									[9].arrDataOut[60]	:=	<0, 8, 0>TIIB(104)^API^Data^io^Outputs^Request Data[30];
									[9].arrDataOut[61]	:=	<0, 8, 8>TIIB(104)^API^Data^io^Outputs^Request Data[30];
									[9].arrDataOut[62]	:=	<0, 8, 0>TIIB(104)^API^Data^io^Outputs^Request Data[31];
									[9].arrDataOut[63]	:=	<0, 8, 8>TIIB(104)^API^Data^io^Outputs^Request Data[31];
									[9].PnIoBoxState 	:=	<0, 16, 0>TIIB(104)^Inputs^PnIoBoxState;
									[10].arrDataIn[0]	:=	<0, 8, 0>TIIB(105)^API^Data^io^Inputs^Response Data[0];
									[10].arrDataIn[1]	:=	<0, 8, 8>TIIB(105)^API^Data^io^Inputs^Response Data[0];
									[10].arrDataIn[2]	:=	<0, 8, 0>TIIB(105)^API^Data^io^Inputs^Response Data[1];
									[10].arrDataIn[3]	:=	<0, 8, 8>TIIB(105)^API^Data^io^Inputs^Response Data[1];
									[10].arrDataIn[4]	:=	<0, 8, 0>TIIB(105)^API^Data^io^Inputs^Response Data[2];
									[10].arrDataIn[5]	:=	<0, 8, 8>TIIB(105)^API^Data^io^Inputs^Response Data[2];
									[10].arrDataIn[6]	:=	<0, 8, 0>TIIB(105)^API^Data^io^Inputs^Response Data[3];
									[10].arrDataIn[7]	:=	<0, 8, 8>TIIB(105)^API^Data^io^Inputs^Response Data[3];
									[10].arrDataIn[8]	:=	<0, 8, 0>TIIB(105)^API^Data^io^Inputs^Response Data[4];
									[10].arrDataIn[9]	:=	<0, 8, 8>TIIB(105)^API^Data^io^Inputs^Response Data[4];
									[10].arrDataIn[10]	:=	<0, 8, 0>TIIB(105)^API^Data^io^Inputs^Response Data[5];
									[10].arrDataIn[11]	:=	<0, 8, 8>TIIB(105)^API^Data^io^Inputs^Response Data[5];
									[10].arrDataIn[12]	:=	<0, 8, 0>TIIB(105)^API^Data^io^Inputs^Response Data[6];
									[10].arrDataIn[13]	:=	<0, 8, 8>TIIB(105)^API^Data^io^Inputs^Response Data[6];
									[10].arrDataIn[14]	:=	<0, 8, 0>TIIB(105)^API^Data^io^Inputs^Response Data[7];
									[10].arrDataIn[15]	:=	<0, 8, 8>TIIB(105)^API^Data^io^Inputs^Response Data[7];
									[10].arrDataIn[16]	:=	<0, 8, 0>TIIB(105)^API^Data^io^Inputs^Response Data[8];
									[10].arrDataIn[17]	:=	<0, 8, 8>TIIB(105)^API^Data^io^Inputs^Response Data[8];
									[10].arrDataIn[18]	:=	<0, 8, 0>TIIB(105)^API^Data^io^Inputs^Response Data[9];
									[10].arrDataIn[19]	:=	<0, 8, 8>TIIB(105)^API^Data^io^Inputs^Response Data[9];
									[10].arrDataIn[20]	:=	<0, 8, 0>TIIB(105)^API^Data^io^Inputs^Response Data[10];
									[10].arrDataIn[21]	:=	<0, 8, 8>TIIB(105)^API^Data^io^Inputs^Response Data[10];
									[10].arrDataIn[22]	:=	<0, 8, 0>TIIB(105)^API^Data^io^Inputs^Response Data[11];
									[10].arrDataIn[23]	:=	<0, 8, 8>TIIB(105)^API^Data^io^Inputs^Response Data[11];
									[10].arrDataIn[24]	:=	<0, 8, 0>TIIB(105)^API^Data^io^Inputs^Response Data[12];
									[10].arrDataIn[25]	:=	<0, 8, 8>TIIB(105)^API^Data^io^Inputs^Response Data[12];
									[10].arrDataIn[26]	:=	<0, 8, 0>TIIB(105)^API^Data^io^Inputs^Response Data[13];
									[10].arrDataIn[27]	:=	<0, 8, 8>TIIB(105)^API^Data^io^Inputs^Response Data[13];
									[10].arrDataIn[28]	:=	<0, 8, 0>TIIB(105)^API^Data^io^Inputs^Response Data[14];
									[10].arrDataIn[29]	:=	<0, 8, 8>TIIB(105)^API^Data^io^Inputs^Response Data[14];
									[10].arrDataIn[30]	:=	<0, 8, 0>TIIB(105)^API^Data^io^Inputs^Response Data[15];
									[10].arrDataIn[31]	:=	<0, 8, 8>TIIB(105)^API^Data^io^Inputs^Response Data[15];
									[10].arrDataIn[32]	:=	<0, 8, 0>TIIB(105)^API^Data^io^Inputs^Response Data[16];
									[10].arrDataIn[33]	:=	<0, 8, 8>TIIB(105)^API^Data^io^Inputs^Response Data[16];
									[10].arrDataIn[34]	:=	<0, 8, 0>TIIB(105)^API^Data^io^Inputs^Response Data[17];
									[10].arrDataIn[35]	:=	<0, 8, 8>TIIB(105)^API^Data^io^Inputs^Response Data[17];
									[10].arrDataIn[36]	:=	<0, 8, 0>TIIB(105)^API^Data^io^Inputs^Response Data[18];
									[10].arrDataIn[37]	:=	<0, 8, 8>TIIB(105)^API^Data^io^Inputs^Response Data[18];
									[10].arrDataIn[38]	:=	<0, 8, 0>TIIB(105)^API^Data^io^Inputs^Response Data[19];
									[10].arrDataIn[39]	:=	<0, 8, 8>TIIB(105)^API^Data^io^Inputs^Response Data[19];
									[10].arrDataIn[40]	:=	<0, 8, 0>TIIB(105)^API^Data^io^Inputs^Response Data[20];
									[10].arrDataIn[41]	:=	<0, 8, 8>TIIB(105)^API^Data^io^Inputs^Response Data[20];
									[10].arrDataIn[42]	:=	<0, 8, 0>TIIB(105)^API^Data^io^Inputs^Response Data[21];
									[10].arrDataIn[43]	:=	<0, 8, 8>TIIB(105)^API^Data^io^Inputs^Response Data[21];
									[10].arrDataIn[44]	:=	<0, 8, 0>TIIB(105)^API^Data^io^Inputs^Response Data[22];
									[10].arrDataIn[45]	:=	<0, 8, 8>TIIB(105)^API^Data^io^Inputs^Response Data[22];
									[10].arrDataIn[46]	:=	<0, 8, 0>TIIB(105)^API^Data^io^Inputs^Response Data[23];
									[10].arrDataIn[47]	:=	<0, 8, 8>TIIB(105)^API^Data^io^Inputs^Response Data[23];
									[10].arrDataIn[48]	:=	<0, 8, 0>TIIB(105)^API^Data^io^Inputs^Response Data[24];
									[10].arrDataIn[49]	:=	<0, 8, 8>TIIB(105)^API^Data^io^Inputs^Response Data[24];
									[10].arrDataIn[50]	:=	<0, 8, 0>TIIB(105)^API^Data^io^Inputs^Response Data[25];
									[10].arrDataIn[51]	:=	<0, 8, 8>TIIB(105)^API^Data^io^Inputs^Response Data[25];
									[10].arrDataIn[52]	:=	<0, 8, 0>TIIB(105)^API^Data^io^Inputs^Response Data[26];
									[10].arrDataIn[53]	:=	<0, 8, 8>TIIB(105)^API^Data^io^Inputs^Response Data[26];
									[10].arrDataIn[54]	:=	<0, 8, 0>TIIB(105)^API^Data^io^Inputs^Response Data[27];
									[10].arrDataIn[55]	:=	<0, 8, 8>TIIB(105)^API^Data^io^Inputs^Response Data[27];
									[10].arrDataIn[56]	:=	<0, 8, 0>TIIB(105)^API^Data^io^Inputs^Response Data[28];
									[10].arrDataIn[57]	:=	<0, 8, 8>TIIB(105)^API^Data^io^Inputs^Response Data[28];
									[10].arrDataIn[58]	:=	<0, 8, 0>TIIB(105)^API^Data^io^Inputs^Response Data[29];
									[10].arrDataIn[59]	:=	<0, 8, 8>TIIB(105)^API^Data^io^Inputs^Response Data[29];
									[10].arrDataIn[60]	:=	<0, 8, 0>TIIB(105)^API^Data^io^Inputs^Response Data[30];
									[10].arrDataIn[61]	:=	<0, 8, 8>TIIB(105)^API^Data^io^Inputs^Response Data[30];
									[10].arrDataIn[62]	:=	<0, 8, 0>TIIB(105)^API^Data^io^Inputs^Response Data[31];
									[10].arrDataIn[63]	:=	<0, 8, 8>TIIB(105)^API^Data^io^Inputs^Response Data[31];
									[10].arrDataOut[0]	:=	<0, 8, 0>TIIB(105)^API^Data^io^Outputs^Request Data[0];
									[10].arrDataOut[1]	:=	<0, 8, 8>TIIB(105)^API^Data^io^Outputs^Request Data[0];
									[10].arrDataOut[2]	:=	<0, 8, 0>TIIB(105)^API^Data^io^Outputs^Request Data[1];
									[10].arrDataOut[3]	:=	<0, 8, 8>TIIB(105)^API^Data^io^Outputs^Request Data[1];
									[10].arrDataOut[4]	:=	<0, 8, 0>TIIB(105)^API^Data^io^Outputs^Request Data[2];
									[10].arrDataOut[5]	:=	<0, 8, 8>TIIB(105)^API^Data^io^Outputs^Request Data[2];
									[10].arrDataOut[6]	:=	<0, 8, 0>TIIB(105)^API^Data^io^Outputs^Request Data[3];
									[10].arrDataOut[7]	:=	<0, 8, 8>TIIB(105)^API^Data^io^Outputs^Request Data[3];
									[10].arrDataOut[8]	:=	<0, 8, 0>TIIB(105)^API^Data^io^Outputs^Request Data[4];
									[10].arrDataOut[9]	:=	<0, 8, 8>TIIB(105)^API^Data^io^Outputs^Request Data[4];
									[10].arrDataOut[10]	:=	<0, 8, 0>TIIB(105)^API^Data^io^Outputs^Request Data[5];
									[10].arrDataOut[11]	:=	<0, 8, 8>TIIB(105)^API^Data^io^Outputs^Request Data[5];
									[10].arrDataOut[12]	:=	<0, 8, 0>TIIB(105)^API^Data^io^Outputs^Request Data[6];
									[10].arrDataOut[13]	:=	<0, 8, 8>TIIB(105)^API^Data^io^Outputs^Request Data[6];
									[10].arrDataOut[14]	:=	<0, 8, 0>TIIB(105)^API^Data^io^Outputs^Request Data[7];
									[10].arrDataOut[15]	:=	<0, 8, 8>TIIB(105)^API^Data^io^Outputs^Request Data[7];
									[10].arrDataOut[16]	:=	<0, 8, 0>TIIB(105)^API^Data^io^Outputs^Request Data[8];
									[10].arrDataOut[17]	:=	<0, 8, 8>TIIB(105)^API^Data^io^Outputs^Request Data[8];
									[10].arrDataOut[18]	:=	<0, 8, 0>TIIB(105)^API^Data^io^Outputs^Request Data[9];
									[10].arrDataOut[19]	:=	<0, 8, 8>TIIB(105)^API^Data^io^Outputs^Request Data[9];
									[10].arrDataOut[20]	:=	<0, 8, 0>TIIB(105)^API^Data^io^Outputs^Request Data[10];
									[10].arrDataOut[21]	:=	<0, 8, 8>TIIB(105)^API^Data^io^Outputs^Request Data[10];
									[10].arrDataOut[22]	:=	<0, 8, 0>TIIB(105)^API^Data^io^Outputs^Request Data[11];
									[10].arrDataOut[23]	:=	<0, 8, 8>TIIB(105)^API^Data^io^Outputs^Request Data[11];
									[10].arrDataOut[24]	:=	<0, 8, 0>TIIB(105)^API^Data^io^Outputs^Request Data[12];
									[10].arrDataOut[25]	:=	<0, 8, 8>TIIB(105)^API^Data^io^Outputs^Request Data[12];
									[10].arrDataOut[26]	:=	<0, 8, 0>TIIB(105)^API^Data^io^Outputs^Request Data[13];
									[10].arrDataOut[27]	:=	<0, 8, 8>TIIB(105)^API^Data^io^Outputs^Request Data[13];
									[10].arrDataOut[28]	:=	<0, 8, 0>TIIB(105)^API^Data^io^Outputs^Request Data[14];
									[10].arrDataOut[29]	:=	<0, 8, 8>TIIB(105)^API^Data^io^Outputs^Request Data[14];
									[10].arrDataOut[30]	:=	<0, 8, 0>TIIB(105)^API^Data^io^Outputs^Request Data[15];
									[10].arrDataOut[31]	:=	<0, 8, 8>TIIB(105)^API^Data^io^Outputs^Request Data[15];
									[10].arrDataOut[32]	:=	<0, 8, 0>TIIB(105)^API^Data^io^Outputs^Request Data[16];
									[10].arrDataOut[33]	:=	<0, 8, 8>TIIB(105)^API^Data^io^Outputs^Request Data[16];
									[10].arrDataOut[34]	:=	<0, 8, 0>TIIB(105)^API^Data^io^Outputs^Request Data[17];
									[10].arrDataOut[35]	:=	<0, 8, 8>TIIB(105)^API^Data^io^Outputs^Request Data[17];
									[10].arrDataOut[36]	:=	<0, 8, 0>TIIB(105)^API^Data^io^Outputs^Request Data[18];
									[10].arrDataOut[37]	:=	<0, 8, 8>TIIB(105)^API^Data^io^Outputs^Request Data[18];
									[10].arrDataOut[38]	:=	<0, 8, 0>TIIB(105)^API^Data^io^Outputs^Request Data[19];
									[10].arrDataOut[39]	:=	<0, 8, 8>TIIB(105)^API^Data^io^Outputs^Request Data[19];
									[10].arrDataOut[40]	:=	<0, 8, 0>TIIB(105)^API^Data^io^Outputs^Request Data[20];
									[10].arrDataOut[41]	:=	<0, 8, 8>TIIB(105)^API^Data^io^Outputs^Request Data[20];
									[10].arrDataOut[42]	:=	<0, 8, 0>TIIB(105)^API^Data^io^Outputs^Request Data[21];
									[10].arrDataOut[43]	:=	<0, 8, 8>TIIB(105)^API^Data^io^Outputs^Request Data[21];
									[10].arrDataOut[44]	:=	<0, 8, 0>TIIB(105)^API^Data^io^Outputs^Request Data[22];
									[10].arrDataOut[45]	:=	<0, 8, 8>TIIB(105)^API^Data^io^Outputs^Request Data[22];
									[10].arrDataOut[46]	:=	<0, 8, 0>TIIB(105)^API^Data^io^Outputs^Request Data[23];
									[10].arrDataOut[47]	:=	<0, 8, 8>TIIB(105)^API^Data^io^Outputs^Request Data[23];
									[10].arrDataOut[48]	:=	<0, 8, 0>TIIB(105)^API^Data^io^Outputs^Request Data[24];
									[10].arrDataOut[49]	:=	<0, 8, 8>TIIB(105)^API^Data^io^Outputs^Request Data[24];
									[10].arrDataOut[50]	:=	<0, 8, 0>TIIB(105)^API^Data^io^Outputs^Request Data[25];
									[10].arrDataOut[51]	:=	<0, 8, 8>TIIB(105)^API^Data^io^Outputs^Request Data[25];
									[10].arrDataOut[52]	:=	<0, 8, 0>TIIB(105)^API^Data^io^Outputs^Request Data[26];
									[10].arrDataOut[53]	:=	<0, 8, 8>TIIB(105)^API^Data^io^Outputs^Request Data[26];
									[10].arrDataOut[54]	:=	<0, 8, 0>TIIB(105)^API^Data^io^Outputs^Request Data[27];
									[10].arrDataOut[55]	:=	<0, 8, 8>TIIB(105)^API^Data^io^Outputs^Request Data[27];
									[10].arrDataOut[56]	:=	<0, 8, 0>TIIB(105)^API^Data^io^Outputs^Request Data[28];
									[10].arrDataOut[57]	:=	<0, 8, 8>TIIB(105)^API^Data^io^Outputs^Request Data[28];
									[10].arrDataOut[58]	:=	<0, 8, 0>TIIB(105)^API^Data^io^Outputs^Request Data[29];
									[10].arrDataOut[59]	:=	<0, 8, 8>TIIB(105)^API^Data^io^Outputs^Request Data[29];
									[10].arrDataOut[60]	:=	<0, 8, 0>TIIB(105)^API^Data^io^Outputs^Request Data[30];
									[10].arrDataOut[61]	:=	<0, 8, 8>TIIB(105)^API^Data^io^Outputs^Request Data[30];
									[10].arrDataOut[62]	:=	<0, 8, 0>TIIB(105)^API^Data^io^Outputs^Request Data[31];
									[10].arrDataOut[63]	:=	<0, 8, 8>TIIB(105)^API^Data^io^Outputs^Request Data[31];
									[10].PnIoBoxState 	:=	<0, 16, 0>TIIB(105)^Inputs^PnIoBoxState;	'}
	fbRFID_Readers				:ARRAY[1..10] OF FB_ID200;
END_VAR

(* stored: Version 1.1.0.1, ProductVersion 3.1.4024.11
   GVL GVL_RFID: Id {97cb121f-e37a-40f2-b9a5-61bf637a8a42} *)
